{attribute 'c++_compatible'}
FUNCTION_BLOCK FB_MyMqtt EXTENDS FB_IotMqttClient
VAR_INPUT
END_VAR
VAR_OUTPUT
END_VAR

VAR
	(* received message *)
	{attribute 'TcEncoding':='UTF-8'}
	sTopicRcv : STRING(255);
	{attribute 'TcEncoding':='UTF-8'}
	sPayloadRcv : STRING(255);
	A: BOOL;
	nVar: INT;
END_VAR

{attribute 'c++_compatible'}
{attribute 'pack_mode' := '4'}
{attribute 'show'}
{attribute 'minimal_input_size' := '4'}
METHOD OnMqttMessage : HRESULT
VAR_IN_OUT CONSTANT
	topic	: STRING;
END_VAR
VAR_INPUT
	payload	: PVOID;
	length	: UDINT;
	qos	: TcIotMqttQos;
	repeated	: BOOL;
END_VAR

VAR
	sRecived: STRING(255);
Test :int ;
END_VAR
SUPER^.nMessagesRcv := SUPER^.nMessagesRcv + 1;

STRNCPY( ADR(sTopicRcv), ADR(topic), SIZEOF(sTopicRcv) );
MEMCPY( ADR(sPayloadRcv), payload, MIN(length, DINT_TO_UDINT(SIZEOF(sPayloadRcv))) );
sTopicRcv;
sPayloadRcv;
nVar := STRING_TO_INT(sPayloadRcv);
IF sTopicRcv = 'BangsareLights' THEN
      CASE nVar OF 
		  0: ;
		  1:  SpotLight := NOT SpotLight;
		  2:  ReceptionLight := NOT ReceptionLight ;
		  3:  EntranceLight := NOT EntranceLight;
		  4:  BedRoomLight := NOT BedRoomLight;
		  5:  Livingroom := NOT Livingroom;
		  6:  WalkingClosett := NOT WalkingClosett;
		  7:  BjornLight := FALSE;
		  8:  BjornLight := TRUE;
		  9:  StairLight := FALSE;
		  10: StairLight := TRUE;
		  11: Spare := NOT Spare;
	  END_CASE
	  	Test :=Test +1;
	END_IF
	sPayloadRcv:='0';
OnMqttMessage := S_OK;
END_METHOD

END_FUNCTION_BLOCK

(* stored: Version 1.1.0.1, ProductVersion 3.1.4024.12
   POU FB_MyMqtt: Id {9c572ae6-e06d-4a20-9a98-0f29ff25b54f}, SpecialFunc None
   Method OnMqttMessage: Id {00b896c3-f44c-4cf4-aba5-b8400ecc5e1a} *)
